{attribute 'linkalways'} 
{attribute 'no_explicit_call' := 'This FB is a CLASS and must be accessed using methods or properties'}
{attribute 'enable_dynamic_creation'}
FUNCTION_BLOCK Node_F_VN_DivideVectorByImage EXTENDS VisionNode
VAR
    aVector : _TcVnVector4_LREAL;
    ipSrcImage : _ITcVnImage;
    ipDestImage : _ITcVnImage;
    hrPrev : _HRESULT(S_OK);
	hresult : _HRESULT(S_OK);
END_VAR

METHOD PUBLIC  Clone : I_Node
VAR
	pNode : POINTER TO Node_F_VN_DivideVectorByImage;
END_VAR
pNode := __NEW(Node_F_VN_DivideVectorByImage);
Clone := pNode^;
END_METHOD

METHOD FB_init : BOOL
VAR_INPUT
	bInitRetains : BOOL; // if TRUE, the retain variables are initialized (warm start / cold start)
	bInCopyCode : BOOL;  // if TRUE, the instance afterwards gets moved into the copy code (online change)
END_VAR
AddInput('aVector', aVector);
AddInput('ipSrcImage', ipSrcImage);
AddInput('hrPrev', hrPrev);
AddOutput('ipDestImage', ipDestImage);
AddOutput('hresult',hresult);
END_METHOD

METHOD PROTECTED OnExecute : HRESULT
hresult.Value := F_VN_DivideVectorByImage(
    aVector := aVector.Value,
    ipSrcImage := ipSrcImage.Value,
	ipDestImage := ipDestImage.Value,
	hrPrev:= hrPrev.Value);
END_METHOD

METHOD PUBLIC PreExecutionCheck
VAR_INPUT
	Check : I_PreExecutionChecks;
END_VAR
Check.IsTrue(ipSrcImage.IsValid, 'ipSrcImage must contain an image');
END_METHOD

END_FUNCTION_BLOCK

(* stored: Version 1.1.0.1, ProductVersion 3.1.4024.13
   POU Node_F_VN_DivideVectorByImage: Id {c3cec74e-ab08-07c7-13fc-44869f258de3}, SpecialFunc None
   Folder Constructor: Id {58b09895-c396-0538-13b0-6812e36ff3fc}
   Method Clone: Id {651f2a09-e38c-0b53-3d72-ec2d13b6d077}
   Method FB_init: Id {26581ad4-634f-0d29-33b2-cb4e7bd577ce}
   Method OnExecute: Id {4e6ee62a-2749-0ff4-2e1c-9569f796d9db}
   Method PreExecutionCheck: Id {dd25991b-6509-03f6-1914-27fa7d4fb46a} *)
